TYPE ST_XBox_Class_Command_Status :
STRUCT
	// Command has been completed
	bDone 	: BOOL;
	// Command is busy
	bBusy 	: BOOL;
	// Command has an error
	bError 	: BOOL;
END_STRUCT
END_TYPE

(* stored: Version 1.1.0.1, ProductVersion 3.1.4024.11
   DUT ST_XBox_Class_Command_Status: Id {76e9dbef-bfd4-4d1b-a378-c1d505289c14} *)
